(* Logix 5000 project; controller OPC_PROJECT vendor 1 type 14 code 89 rev 20.19; software revision 20.05 *)

TASK Diag_Task (periodic, rate 500 ms, priority 10, watchdog 500 ms) : Diag_Program   // Periodic diagnostic task (GSV, FaultLog, Modules)
TASK MainTask (continuous, watchdog 500 ms) : MainProgram

MODULES
   Controller : vendor 1 type 14 code 89 (CompactLogixL23E_QBFC1_Controller 0, rev 20.19)
      LocalENB : vendor 1 type 12 code 191 (CompactLogixL23E_QBFC1_Ethernet 1, rev 20.11)
      Local : CompactBus (CompactVirtualAdapter 3, rev 20.11)
         Discrete_Inputs : vendor 1 type 7 code 320 (Compact 1, rev 3.1, Input RPI 20 ms)
         Discrete_Outputs : vendor 1 type 7 code 322 (Compact 2, rev 3.1, Output RPI 20 ms)
         Analog_IO : vendor 1 type 10 code 120 (Compact 3, rev 1.1, Output RPI 80 ms)
         Counters : vendor 1 type 109 code 70 (Compact 4, rev 1.1, Output RPI 20 ms)
END_MODULES

PROGRAM Diag_Program   (* main routine Diagnostic_Routine *)
VAR
   DIAG_ControllerStatus : INT;
   DIAG_CPU_Fault : BOOL;
   DIAG_CPU_Local : BOOL;
   DIAG_CPU_MajorFault : ALIAS FOR DIAG_ControllerStatus.11;
   DIAG_CPU_MinorFault : ALIAS FOR DIAG_ControllerStatus.10;
   DIAG_CPU_Remote : BOOL;
   DIAG_CPU_Warning : BOOL;
   DIAG_IOLedStatus : INT;
   DIAG_MajorEvents : INT;
   DIAG_MajorFaultBits : DINT;
   DIAG_MF_ConfigFault : ALIAS FOR DIAG_MajorFaultBits.4;
   DIAG_MF_IOFault : ALIAS FOR DIAG_MajorFaultBits.3;
   DIAG_MF_MemoryFault : ALIAS FOR DIAG_MajorFaultBits.5;
   DIAG_MF_ModuleMismatch : ALIAS FOR DIAG_MajorFaultBits.8;
   DIAG_MF_NonRecoverable : ALIAS FOR DIAG_MajorFaultBits.2;
   DIAG_MF_PowerLoss : ALIAS FOR DIAG_MajorFaultBits.0;
   DIAG_MF_Watchdog : ALIAS FOR DIAG_MajorFaultBits.6;
   DIAG_MOD_EntryStatus : INT;
   DIAG_MOD_FaultCode : INT;
   DIAG_MOD_FaultInfo : DINT;
   DIAG_MOD_Mode : DINT;
   DIAG_ProductCode : INT;
   DIAG_ProductRev : INT;
   DIAG_SerialNumber : DINT;
END_VAR

ROUTINE Diagnostic_Routine   (* structured text *)
   // CPU / ControllerDevice
   GSV(CONTROLLERDEVICE, , ProductCode,   DIAG_ProductCode);
   GSV(CONTROLLERDEVICE, , ProductRev,    DIAG_ProductRev);
   GSV(CONTROLLERDEVICE, , SerialNumber,  DIAG_SerialNumber);
   GSV(CONTROLLERDEVICE, , Status,        DIAG_ControllerStatus);
   
   // FaultLog
   GSV(FAULTLOG, , MajorEvents,     DIAG_MajorEvents);
   GSV(FAULTLOG, , MajorFaultBits,  DIAG_MajorFaultBits);
   
   // I/O LED Global
   GSV(MODULE, , LEDStatus, DIAG_IOLedStatus);
   
   
   DIAG_CPU_Remote := DIAG_ControllerStatus.13 AND DIAG_ControllerStatus.12;
   
   DIAG_CPU_Local := NOT DIAG_CPU_Remote;
   DIAG_CPU_Fault := DIAG_ControllerStatus.7 OR DIAG_ControllerStatus.11;
   
   DIAG_CPU_Warning := DIAG_ControllerStatus.10 AND (NOT DIAG_CPU_Fault);
   
   
END_ROUTINE
END_PROGRAM

PROGRAM MainProgram   (* main routine MainRoutine *)

ROUTINE MainRoutine   (* ladder *)
END_ROUTINE
END_PROGRAM
